Fanuc KAREL source: KS00036.KL

PROGRAM KS00036
%NOLOCKGROUP
TYPE
  REC_T = STRUCTURE
    VALUE: INTEGER
    FLAG: BOOLEAN
  ENDSTRUCTURE
VAR
  A: ARRAY[4] OF POSITION
  B: ARRAY[4] OF POSITION
  FLAG: BOOLEAN
  N: INTEGER
  STATUS: INTEGER
  PN: STRING[80]
  VN: STRING[80]
BEGIN
  PN = ''
  VN = 'A'
  FLAG = A = B
END KS00036
